PROGRAM MAIN
VAR
    bInit : BOOL := TRUE; 
    bSend : BOOL := TRUE; 

    fbMsg : FB_TcMessage; 
END_VAR

IF bInit THEN
	bInit := FALSE;
	fbMsg.CreateEx(TC_Events.AlarmsAndEvents.Estop, 0);
END_IF

IF bSend THEN
	bSend := FALSE;
	fbMsg.Send(0);
	
END_IF

END_PROGRAM

(* stored: Version 1.1.0.1, ProductVersion 3.1.4024.12
   POU MAIN: Id {bb22a364-aba9-4699-8efd-cb42e3362f0a}, SpecialFunc None *)
